// TIA Portal V20 export
TYPE "PLC_STATUS_UDT"
   STRUCT
      RUN_STOP : Int;   // RUN/STOP LED (Yellow/Green) / 运行/停止 LED (黄/Green)
      ER_ERROR : Int;   // ERROR LED (Red) / 错误 LED (红)
      MT_MAINT : Int;   // MAINT LED (Yellow) / MAINT LED (黄)
      QSTATUS : Bool;   // FAIL SAFE STATUS / 安全失败 状态
      RIOforFA_VALUE_STATUS : Bool;   // FAIL SAFE STATUS / 安全失败 状态
      F_DEVICE_PASSIVATED : Bool;   // FAIL SAFE STATUS / 安全失败 状态
   END_STRUCT;
END_TYPE
